// TIA Portal V18 export
// export: Created 2026-06-08T16:04:36.6826527Z, ExportSetting WithDefaults, DisplayName Totally Integrated Automation Portal, DisplayVersion V18, DisplayName TIA Portal Openness, DisplayVersion V18, DisplayName TIA Portal Version Control Interface, DisplayVersion V18, DisplayName STEP 7 Professional, DisplayVersion V18, DisplayName STEP 7 Safety, DisplayVersion V18, DisplayName WinCC Professional, DisplayVersion V18
VAR_GLOBAL   // PLC tag table "INPUT"
   I_Mode AT %I0.0 : Bool;   // Switch chế độ 1 auto, 0 manu
   I_CB_Cao AT %I0.1 : Bool;   // Cảm biến sản phẩm cao
   I_CB_Trung_Binh AT %I0.2 : Bool;   // Cảm biến sản phẩm trung bình
   I_CB_Thap AT %I0.3 : Bool;   // Cảm biến sản phẩm thấp
   I_BT AT %I0.4 : Bool;   // Chạy/Dừng động cơ băng tải
   I_Xylanh_Cao AT %I0.5 : Bool;   // Đóng/mở xi lanh sản phẩm cao
   I_Xylanh_TB AT %I0.6 : Bool;   // Đóng/mở xi lanh sản phẩm trung bình
END_VAR
